FUNCTION_BLOCK FB_MasterCart
VAR
	//  IO and check
	m_endoScopePedalIO AT%I* :BOOL;
	m_endoScopeIOCheck :FB_IOCheck;
	
	m_clutchPedalIO AT%I* :BOOL;
	m_clutchIOCheck :FB_IOCheck;
	
	m_surgonHeadInIO AT%I* :BOOL;
	m_headInCheck:FB_IOCheck;
	
	m_armSwitchIO AT%I* :BOOL;
	m_armSwitchCheck:FB_IOToggleCheck;
	
	m_electricCutLeft AT %I* :BOOL;
	m_electricCutLeftAllow AT %I* :BOOL;
	
	m_electricCutRight AT %I* :BOOL;
	m_electricCutRightAllow AT %I* :BOOL;
	
	m_electricCoagulLeft AT %I* :BOOL;
	m_electricCoagulLeftAllow AT %I* :BOOL;
	
	m_electricCoagulRight AT %I* :BOOL;
	m_electricCoagulRightAllow AT %I* :BOOL;
	
	m_elecKnifeCtrlWord AT %Q* :DINT;
	
	// cart status
	m_cartStatus  : ST_CartStatus;
	
	// cart joints
	// [monitor lift, monitor rotate, armset, pedal]
	m_cartJoints:ARRAY[1..4] OF FB_CartJoint;
	
	// cart joint motion control IO
	//[monitor_up, monitor_down, monitor_cwRotate, monitor_ccwRotate, armset_up, armset_down, pedal_in, pedal_out]
	m_cartJointCtrlIO AT%I* :ARRAY[1..8] OF BOOL ;
	m_cartJointCtrlIOCheck :ARRAY[1..8] OF FB_IOCheck;
	
	//electrotome control io
	m_electricCutLeftOn :BOOL;
	m_electricCutRightOn :BOOL;
	m_electricCoagulLeftOn : BOOL;
	m_electricCoagulRightOn : BOOL;
	//Triggering several energies at once
	m_eleCtrlState : UINT;
	//The type of instrument energy of the master hand corresponding to the slave hand
	m_energyType :ARRAY[1..g_mArmNum] OF UINT :=[2(0)];
	
	// cart joint control data
	m_jntEnableCounts:Vec4i ;
	m_jntDisableCounts:Vec4i ;
	m_jntEnableCountsThres:INT:=500;
	m_jntCmdMotionDir :Vec4i;
	m_cmdJntTrq :Vec4d;
	m_cmdJntPos :Vec4d;
	m_cmdJntVel :Vec4d;
	m_jntEnableFlag :Vec4b;
	
	//cart ergonomic adjust data
	m_UIData : ST_CartUIData;
	m_carInMotion : INT; // 0:  no mition, 1: mamual adjust, 2: ergonomic adjust
	m_jntSoftwareLimit :ARRAY [1..4] OF LREAL := [0.001, 1*g_deg2Rad, 0.001, 0.001];
	m_cmdArrival : Vec4b;
	
	// cart joint status data
	m_curMotorPos :Vec4d;
	m_curLinkPos :Vec4d;
	m_curJntPos :Vec4d;
	m_curJntVel :Vec4d;
	m_curJntTrq :Vec4d;
	m_rawJntCurrent :Vec4d;
	m_filtJntCurrent :Vec4d;
	m_cmdJntCurrent : Vec4d;

END_VAR

METHOD eleKnifeCtrl : DINT
VAR_IN_OUT CONSTANT
	m_armState:ARRAY[1..g_mArmNum] OF E_masterArmState ;
	m_teleSlaveArmIdx :ARRAY[1..g_mArmNum] OF E_MatchedSlaveArmIdx;
	m_instruStauts: ARRAY[1..g_sArmNum] OF ST_InstruStatus;
END_VAR
//Foot trigger check
m_electricCutLeftOn := m_electricCutLeft AND m_electricCutLeftAllow AND m_armState[1] = MasterArmState_MasterSlave ;
m_electricCutRightOn := m_electricCutRight AND m_electricCutRightAllow AND m_armState[2] = MasterArmState_MasterSlave ;
m_electricCoagulLeftOn := m_electricCoagulLeft AND m_electricCoagulLeftAllow AND m_armState[1] = MasterArmState_MasterSlave ;
m_electricCoagulRightOn := m_electricCoagulRight AND m_electricCoagulRightAllow AND m_armState[2] = MasterArmState_MasterSlave ;

//You cannot excite two energies at the same time
m_eleCtrlState := BOOL_TO_UINT(m_electricCutLeftOn) + BOOL_TO_UINT(m_electricCutRightOn)
										 + BOOL_TO_UINT(m_electricCoagulLeftOn) + BOOL_TO_UINT(m_electricCoagulRightOn);

IF m_teleSlaveArmIdx[1] > 0 THEN
	m_energyType[1] := m_instruStauts[m_teleSlaveArmIdx[1]].m_energyType;
	m_energyType[2] := m_instruStauts[m_teleSlaveArmIdx[2]].m_energyType;
END_IF

IF m_eleCtrlState = 1 THEN
	IF (m_electricCutLeftOn AND  m_energyType[1] = InstruType_isMonopole) OR (m_electricCutRightOn AND  m_energyType[2] = InstruType_isMonopole) THEN
		eleKnifeCtrl := EnergyCtrlWord_isMonopoleCut;
	ELSIF (m_electricCoagulLeftOn AND m_energyType[1] = InstruType_isMonopole) OR (m_electricCoagulRightOn AND  m_energyType[2] = InstruType_isMonopole) THEN
		eleKnifeCtrl := EnergyCtrlWord_isMonopoleCoagul;
	ELSIF (m_electricCoagulLeftOn AND m_energyType[1] = InstruType_isBipolar) OR (m_electricCoagulRightOn AND  m_energyType[2] = InstruType_isBipolar) THEN
		eleKnifeCtrl := EnergyCtrlWord_isBipolarCoagul;
	ELSIF (m_electricCutLeftOn AND m_energyType[1] = InstruType_isUltraKnife) OR (m_electricCutRightOn AND  m_energyType[2] = InstruType_isUltraKnife) THEN
		eleKnifeCtrl := EnergyCtrlWord_isUltraMin;
	ELSIF (m_electricCoagulLeftOn AND m_energyType[1] = InstruType_isUltraKnife) OR (m_electricCoagulRightOn AND  m_energyType[2] = InstruType_isUltraKnife) THEN
		eleKnifeCtrl := EnergyCtrlWord_isUltraMax;
		
	ELSE
		eleKnifeCtrl := EnergyCtrlWord_NoOutput;
	END_IF
ELSE
	eleKnifeCtrl := EnergyCtrlWord_NoOutput;
END_IF
END_METHOD

METHOD ergonomicAdjust : INT
VAR_INPUT
END_VAR
VAR
	i : INT;
	err:Vec4d;
END_VAR
vecSub(m_UIData.m_cmdJntPos,m_curJntPos, err);
ergonomicAdjust := 2;
//only update command after joints is truly enabled
FOR i := 1 TO 4 DO
	IF m_jntEnableFlag[i] AND m_cartJoints[i].isEnabled() AND m_jntEnableCounts[i]>= m_jntEnableCountsThres THEN
		m_cmdJntVel[i]:=sign(m_UIData.m_cmdJntPos[i]-m_cartJoints[i].jntPos)*(GVL_CartJointParameters.g_jntCtrlMotionVel[i]);
		IF ABS(err[i]) < m_jntSoftwareLimit[i]/3 THEN
			m_cmdJntVel[i]:=0;
		END_IF
		m_cmdJntPos[i] := LIMIT(GVL_CartJointParameters.g_minJntPos[i] + m_jntSoftwareLimit[i],  m_cmdJntPos[i] + m_cmdJntVel[i]*g_cartCtrlCycleTime, GVL_CartJointParameters.g_maxJntPos[i] - m_jntSoftwareLimit[i]);
	
	ELSE
		m_cmdJntVel[i]:=0;
		m_cmdJntPos[i] := m_cartJoints[i].jntPos;
	END_IF	
END_FOR
END_METHOD

METHOD PUBLIC getStatus : BOOL
VAR_IN_OUT
	// cart status data
	r_cartStatus :ST_CartStatus;
	
	// cart joint data
	r_cartJointData :ST_CartJointData;
	
END_VAR
r_cartStatus := m_cartStatus;


// current joint data
r_cartJointData.m_curMotorPos:=m_curMotorPos;
r_cartJointData.m_curLinkPos:=m_curLinkPos;
r_cartJointData.m_curJntPos:=m_curJntPos;
r_cartJointData.m_curJntVel:=m_curJntVel;
r_cartJointData.m_curJntTrq:=m_curJntVel;
r_cartJointData.m_rawJntCurrent:=m_rawJntCurrent;
r_cartJointData.m_filtJntCurrent:=m_filtJntCurrent;

// command joint data
r_cartJointData.m_cmdJntPos:=m_cmdJntPos;
r_cartJointData.m_cmdJntVel:=m_cmdJntVel;
r_cartJointData.m_cmdJntTrq:=m_cmdJntTrq;
r_cartJointData.m_cmdJntCurrent:=m_cmdJntCurrent;
END_METHOD

METHOD PUBLIC init : BOOL
VAR_INPUT
END_VAR
VAR
	i:INT;
	initLinkPos :LREAl;
END_VAR
// joint init
FOR i:=1 TO 4 DO
	m_cartJoints[i].init(i,g_cartCtrlCycleTime);
	m_cartJoints[i].initJntPos();
END_FOR

// motor and link encoder of  monitor rotation are on different  joints
// transfer monitor angle from link side to motor side
initLinkPos:= monitorAngLink2Motor(m_cartJoints[2].initLinkPos);
m_cartJoints[2].initJntPosReset(initLinkPos);

// init commands
FOR i:=1 TO 4 DO
	m_jntEnableCounts[i]:=0;
	m_jntDisableCounts[i]:=0;
	m_jntEnableFlag[i]:=FALSE;
	m_jntCmdMotionDir[i]:=0;
	m_cmdJntTrq[i]:=0;
	m_cmdJntVel[i]:=0;
	m_cmdJntPos[i]:=m_cartJoints[i].jntPos;
END_FOR

m_cartStatus.m_initFlag :=true;
END_METHOD

METHOD manualAdjust : INT
VAR_INPUT
END_VAR
VAR
	i : INT;
END_VAR
// update joint command positon
manualAdjust := 1;
//only update command after joints is truly enabled
FOR i := 1 TO 4 DO
	IF  m_jntEnableFlag[i] AND m_cartJoints[i].isEnabled() AND m_jntEnableCounts[i]>= m_jntEnableCountsThres THEN
		//  update command joint velocity
		m_cmdJntVel[i]:=m_jntCmdMotionDir[i]*GVL_CartJointParameters.g_jntCtrlMotionVel[i];
		
		// limit handle
		IF (m_cmdJntPos[i]> GVL_CartJointParameters.g_maxJntPos[i] - m_jntSoftwareLimit[i] AND m_cmdJntVel[i] >0 ) OR 
				(m_cmdJntPos[i]< GVL_CartJointParameters.g_minJntPos[i] + m_jntSoftwareLimit[i] AND m_cmdJntVel[i] <0 )  THEN
				m_cmdJntVel[i] := 0.0;
		END_IF
		m_cmdJntPos[i]:= m_cmdJntPos[i]+ m_cmdJntVel[i]*g_cartCtrlCycleTime;
	ELSE
		m_cmdJntVel[i]:=0;
		m_cmdJntPos[i] := m_cartJoints[i].jntPos;
	END_IF
END_FOR
END_METHOD

// TODO
METHOD PROTECTED monitorAngLink2Image : LREAL
VAR_INPUT
	i_linkPos:LREAL;
END_VAR
VAR
	A,B,C,D,E,F,G,H,I,X0,X1,X2,X3,X4,X5,X6,X7,X8,X9,X10,X11,X12,Z0:LREAL;	
END_VAR

X0:=i_linkPos;  //监视器旋转

A:=227; B:=216; C:=159.285; D:=150.297; E:=195; F:=130; G:=137; H:=40; I:=99;
X4:=ATAN(H/I); X5:=ATAN(F/G);
X8:=SQRT(F*F+G*G);
X12:=sqrt(H*H+I*I);
X9:=sqrt(E*E+X12*X12-2*E*X12*cos(X0));
X6:=acos((B*B+X8*X8-X9*X9)/(2*B*X8));
X10:=acos((B*B+X9*X9-X8*X8)/(2*B*X9));
X11:=acos((X9*X9+X12*X12-E*E)/(2*X9*X12));
X7:=X10+X11;
X2:=X5-X6;
X3:=pi-X7+X2;
X1:=X3-X4;

monitorAngLink2Image:=X1;
END_METHOD

// TODO
METHOD PROTECTED monitorAngLink2Motor : LREAL
VAR_INPUT
	i_linkPos:LREAL;
END_VAR
VAR
	A,B,C,D,E,F,G,H,I,X0,X1,X2,X3,X4,X5,X6,X7,X8,X9,X10,X11,X12,Z0:LREAL;	
END_VAR

X0:=i_linkPos;  //监视器旋转

A:=227; B:=216; C:=159.285; D:=150.297; E:=195; F:=130; G:=137; H:=40; I:=99;
X4:=ATAN(H/I); X5:=ATAN(F/G);
X8:=SQRT(F*F+G*G);
X12:=sqrt(H*H+I*I);
X9:=sqrt(E*E+X12*X12-2*E*X12*cos(X0));
X6:=acos((B*B+X8*X8-X9*X9)/(2*B*X8));
X10:=acos((B*B+X9*X9-X8*X8)/(2*B*X9));
X11:=acos((X9*X9+X12*X12-E*E)/(2*X9*X12));
X7:=X10+X11;
X2:=X5-X6;
X3:=pi-X7+X2;
X1:=X3-X4;

monitorAngLink2Motor:=X2;
END_METHOD

//TODO
METHOD PROTECTED monitorAngMotor2Link : LREAL
VAR_INPUT
	i_motorPos:LREAL;
END_VAR
VAR
	A,B,C,D,E,F,G,H,I,X0,X1,X2,X3,X4,X5,X6,X7,X8,X9,X10,X11,X12,Z0:LREAL;	
END_VAR
X2:=i_motorPos;

A:=227; B:=216; C:=159.285; D:=150.297; E:=195; F:=130; G:=137; H:=40; I:=99;
X5:=atan(F/G);
X6:=X5-X2;
X8:=sqrt(F*F+G*G);
X9:=sqrt(B*B+X8*X8-2*B*X8*cos(X6));
X12:=SQRT(H*H+I*I);
X0:=ACOS((E*E+X12*X12-X9*X9)/(2*E*X12));

monitorAngMotor2Link:=X0;
END_METHOD

METHOD reachUITargetCheck : bool
VAR
	i :INT;
	err:Vec4d;
END_VAR
vecSub(m_UIData.m_cmdJntPos,m_curJntPos, err);

// joint error check
FOR i:=1 TO 4 DO 
	m_cmdArrival[i] :=  ABS(err[i]) < m_jntSoftwareLimit[i]/2;
END_FOR
END_METHOD

METHOD PUBLIC run : BOOL
VAR_IN_OUT CONSTANT
	i_cartUIData : ST_CartUIData;
END_VAR
VAR
	i:INT;
END_VAR
// update IO signals
updateIO(i_cartUIData);

// update cart status
updateStatus();

// update controller and command
updateCmds();

// send command to joint driver
FOR i:=1 TO 4 DO
	// joint enable
	IF m_jntEnableFlag[i] AND NOT(SafetyCheck.m_safetyCheckData.m_cartErrFlag[i]) AND MasterArmControl.m_masterStatus.m_armState[1] <> MasterArmState_MasterSlave 
								AND MasterArmControl.m_masterStatus.m_armState[2] <> MasterArmState_MasterSlave THEN
		m_cartJoints[i].enable();
	ELSE
		m_cartJoints[i].disable();
	END_IF
	
	// set command position
	m_cartJoints[i].updateCmds(DriverOPMode_Pos,m_cmdJntPos[i],m_cmdJntTrq[i]);
END_FOR
END_METHOD

PROPERTY status : ST_CartStatus
GET
status := m_cartStatus;
END_GET
END_PROPERTY

METHOD PROTECTED updateCmds : BOOL
VAR_INPUT
END_VAR
VAR
	i:INT;
	
END_VAR
IF (m_jntCmdMotionDir[1] <>0 OR m_jntCmdMotionDir[2]<>0 OR m_jntCmdMotionDir[3] <>0 OR m_jntCmdMotionDir[4] <>0) AND m_carInMotion <> 2 THEN
	m_carInMotion := manualAdjust();
ELSIF (m_UIData.m_ergonomicCrl.m_recovErgonEnable OR m_UIData.m_ergonomicCrl.m_cancelRecovErgonEnable) AND m_carInMotion <> 1 THEN
	m_carInMotion := ergonomicAdjust();
ELSE
	m_carInMotion := 0;
END_IF

reachUITargetCheck();
IF m_cmdArrival[1] AND m_cmdArrival[2] AND m_cmdArrival[3] AND m_cmdArrival[4] THEN
	IF m_UIData.m_ergonomicCrl.m_recovErgonEnable THEN
		m_cartStatus.m_cancelErgonAdjustArrival := FALSE;
		m_cartStatus.m_ergonAdjustArrival := TRUE;
	END_IF
	IF m_UIData.m_ergonomicCrl.m_cancelRecovErgonEnable THEN
		m_cartStatus.m_ergonAdjustArrival := FALSE;
		m_cartStatus.m_cancelErgonAdjustArrival := TRUE;
	END_IF
ELSE
	m_cartStatus.m_ergonAdjustArrival := FALSE;
	IF m_UIData.m_ergonomicCrl.m_recovErgonEnable THEN
		m_cartStatus.m_cancelErgonAdjustArrival := FALSE;
	END_IF
END_IF
END_METHOD

METHOD PROTECTED updateIO : BOOL
VAR_INPUT
	i_cartUIData : ST_CartUIData;
END_VAR
VAR
	i:INT;
	idxOffset:INT;
END_VAR
// updata IO signals
m_cartStatus.m_clutchSwitch:= m_clutchIOCheck.check(m_clutchPedalIO);
m_cartStatus.m_endoscopeSwitch := m_endoScopeIOCheck.check(m_endoScopePedalIO);
m_cartStatus.m_surgonReady := m_headInCheck.check(m_surgonHeadInIO);
m_cartStatus.m_armSwitch :=m_armSwitchCheck.check(m_armSwitchIO);
m_UIData := i_cartUIData;

//updata Electrotome control
m_elecKnifeCtrlWord := eleKnifeCtrl(MasterArmControl.m_masterStatus.m_armState , MasterArmControl.m_masterStatus.m_teleSlaveArmIdx , MasterArmControl.m_masterInputDataPool.m_slaveStatus.m_instruStauts );

//updata pedal hover and pedal trigger
m_cartStatus. m_pedalHover[1] := m_electricCutLeftAllow OR m_electricCoagulLeftAllow;
m_cartStatus. m_pedalHover[2] := m_electricCutRightAllow OR m_electricCoagulRightAllow;
IF m_electricCutLeftOn AND m_eleCtrlState = 1 THEN
	m_cartStatus.m_electricKnifePedalTrigger[1] := 1;
ELSIF m_electricCoagulLeftOn AND m_eleCtrlState = 1 THEN
	m_cartStatus.m_electricKnifePedalTrigger[1] := 2;
ELSE
	m_cartStatus.m_electricKnifePedalTrigger[1] := 0;
END_IF

IF m_electricCutRightOn AND m_eleCtrlState = 1 THEN
	m_cartStatus.m_electricKnifePedalTrigger[2] := 1;
ELSIF m_electricCoagulRightOn AND m_eleCtrlState = 1 THEN
	m_cartStatus.m_electricKnifePedalTrigger[2] := 2;
ELSE
	m_cartStatus.m_electricKnifePedalTrigger[2] := 0;
END_IF

//update cart joint control switch
FOR i:=1 TO 4 DO 
	idxOffset:= 2*(i-1);
	IF m_cartJointCtrlIOCheck[1+idxOffset].check(m_cartJointCtrlIO[1+idxOffset]) THEN
		m_jntCmdMotionDir[i]:=1;
	ELSIF  m_cartJointCtrlIOCheck[2+idxOffset].check(m_cartJointCtrlIO[2+idxOffset]) THEN
		m_jntCmdMotionDir[i]:=-1;
	ELSE
		m_jntCmdMotionDir[i]:=0;
	END_IF
END_FOR


// if console is already in motion, only check the currently moving joint
IF m_cartStatus.m_consoleInAdjust THEN
	FOR i:=1 TO 4 DO
		IF NOT(m_cartJoints[i].isEnabled()) THEN
			m_jntCmdMotionDir[i] := 0;
		END_IF
	END_FOR
END_IF


// update joint enable flag
FOR i:= 1 TO 4 DO
	IF m_jntCmdMotionDir[i] <> 0 OR m_UIData.m_ergonomicCrl.m_recovErgonEnable OR m_UIData.m_ergonomicCrl.m_cancelRecovErgonEnable THEN
		m_jntEnableFlag[i] := TRUE;
		m_jntEnableCounts[i]:= LIMIT(0, m_jntEnableCounts[i]+1, m_jntEnableCountsThres);
		m_jntDisableCounts[i]:=m_jntEnableCountsThres;
	ELSE
		m_jntEnableCounts[i]:=0;
		m_jntDisableCounts[i]:= LIMIT(0, m_jntDisableCounts[i]-1, m_jntEnableCountsThres);
		m_jntEnableFlag[i] :=m_jntDisableCounts[i]>0; 
	END_IF
END_FOR

// Do not adjust during master-slave control
IF MasterArmControl.m_masterStatus.m_armState[1] = MasterArmState_MasterSlave OR MasterArmControl.m_masterStatus.m_armState[1] = MasterArmState_Endoscope OR
	MasterArmControl.m_masterStatus.m_armState[2] = MasterArmState_MasterSlave OR MasterArmControl.m_masterStatus.m_armState[2] = MasterArmState_Endoscope  THEN
	m_jntCmdMotionDir := g_zeroVec4i;
END_IF
END_METHOD

METHOD PROTECTED updateStatus : BOOL
VAR_INPUT
END_VAR
VAR
	i:INT;
END_VAR
// update cart joints status
FOR i:=1  TO 4 DO
	m_cartJoints[i].updateStatus();
END_FOR

// get joint data
FOR i:=1 TO 4 DO
	m_curMotorPos[i]:=m_cartJoints[i].motorPos;
	m_curLinkPos[i]:=m_cartJoints[i].linkPos;
	m_curJntPos[i]:=m_cartJoints[i].jntPos;
	m_curJntVel[i]:=m_cartJoints[i].jntVel;
	m_curJntTrq[i]:=m_cartJoints[i].jntTrq;
	m_rawJntCurrent[i]:=m_cartJoints[i].rawCurrent;
	m_filtJntCurrent[i]:=m_cartJoints[i].filtCurrent;
	m_cmdJntCurrent[i]:=m_cartJoints[i].cmdCurrent;
END_FOR 

// transfer monitor angle from link side to motor side
m_curLinkPos[2]:= monitorAngLink2Motor(m_cartJoints[2].linkPos);

// get monitor angle
m_cartStatus.m_monitorAngle:= monitorAngLink2Image(m_cartJoints[2].linkPos);

// check if cart in motion
m_cartStatus.m_consoleInAdjust:=FALSE;
FOR i:=1 TO 4 DO
	IF m_cartJoints[i].isEnabled() THEN
		m_cartStatus.m_consoleInAdjust:=TRUE;
		EXIT;
	END_IF
END_FOR

// check if monitor in motion
m_cartStatus.m_monitorInAdjust:=m_cartJoints[2].isEnabled();

// check if cart in manual adjustment
m_cartStatus.m_consoleInManualAdjust := FALSE;
FOR i:=1 TO 4 DO
	IF m_jntCmdMotionDir[i] <> 0 AND m_cartJoints[i].isEnabled() THEN
		m_cartStatus.m_consoleInManualAdjust := TRUE;
		EXIT;
	END_IF
END_FOR
END_METHOD

END_FUNCTION_BLOCK

(* stored: Version 1.1.0.1, ProductVersion 3.1.4024.12
   POU FB_MasterCart: Id {05baaa0e-c853-48bc-a37c-d593cfa5bf2b}, SpecialFunc None
   Folder property: Id {37b9f91a-fbe1-4cae-807d-574d49e247d7}
   Method eleKnifeCtrl: Id {802e30d4-05e6-4f42-9cf9-00572025b770}
   Method ergonomicAdjust: Id {2e585813-8b6a-4acc-85dd-29e49a47183d}
   Method getStatus: Id {3f39e291-1358-48a2-aa04-62d9bb4689e3}
   Method init: Id {a9830b95-e937-4a29-b70e-785e20452d37}
   Method manualAdjust: Id {9030940b-1f5c-4fe8-8e49-9b86403f7e35}
   Method monitorAngLink2Image: Id {3a8f7b3f-992a-495f-9594-efaf7000460f}
   Method monitorAngLink2Motor: Id {be375282-cfa2-4973-91da-b3215777ab52}
   Method monitorAngMotor2Link: Id {5a608b24-1792-4091-9318-b2f1f860af4d}
   Method reachUITargetCheck: Id {58f1d629-33ee-4e90-90f3-a5c453c13e46}
   Method run: Id {5adedbe6-c484-4199-b427-bc8af7c6d1b0}
   Property status: Id {cd2a750f-147a-42a5-85cd-a7d5a815c963}
   Get Get: Id {c1788322-40e1-4e3e-a26b-a8239c1e1e6d}
   Method updateCmds: Id {a083537e-6f52-4b88-8b83-3c9a5d0db87a}
   Method updateIO: Id {2eedbee2-a8d4-4513-b19a-4a2795c7d360}
   Method updateStatus: Id {7dc0698e-0910-43df-8937-4fb176791915} *)
